// TIA Portal V17 export
// export: Created 2022-06-16T09:21:07.0995622Z, ExportSetting WithDefaults, DisplayName Totally Integrated Automation Portal, DisplayVersion V17, DisplayName TIA Portal Openness, DisplayVersion V17, DisplayName TIA Portal Version Control Interface, DisplayVersion V17, DisplayName STEP 7 Professional, DisplayVersion V17, DisplayName STEP 7 Safety, DisplayVersion V17, DisplayName WinCC Advanced, DisplayVersion V17
DATA_BLOCK "projectParam"   // DB1
{ S7_Optimized_Access := 'TRUE' }
VERSION : 0.1
// stored: AutoNumber true, DBAccessibleFromOPCUA true, IsOnlyStoredInLoadMemory false, IsRetainMemResEnabled false, IsWriteProtectedInAS false, MemoryReserve 100
   VAR
      armParams : Array[1..3] of "typeArmParam";
   END_VAR
BEGIN
   armParams[1..3].armType := 'RCMA';
   armParams[1..3].armGeom.outLength := 8.839;
   armParams[1..3].armGeom.inLength := 9.449;
   armParams[1..3].armGeom.brHeight := 10.47;
   armParams[2].armGeom.brWidth := 10.47;
   armParams[1].motionControlParam.angleInputParam.filterTimeConsts[1..3] := 0.1;
   armParams[2].motionControlParam.angleInputParam.filterTimeConsts[1..3] := 0.1;
   armParams[3].motionControlParam.angleInputParam.filterTimeConsts[1..3] := 0.1;
   armParams[1].motionControlParam.angleInputParam.scalingParams[1].axisNum := 1;
   armParams[1].motionControlParam.angleInputParam.scalingParams[2].axisNum := 2;
   armParams[1].motionControlParam.angleInputParam.scalingParams[3].axisNum := 3;
   armParams[2].motionControlParam.angleInputParam.scalingParams[1].axisNum := 1;
   armParams[2].motionControlParam.angleInputParam.scalingParams[2].axisNum := 2;
   armParams[2].motionControlParam.angleInputParam.scalingParams[3].axisNum := 3;
   armParams[3].motionControlParam.angleInputParam.scalingParams[1].axisNum := 1;
   armParams[3].motionControlParam.angleInputParam.scalingParams[2].axisNum := 2;
   armParams[3].motionControlParam.angleInputParam.scalingParams[3].axisNum := 3;
   armParams[1].motionControlParam.angleInputParam.scalingParams[1..3]."a" := 1.0;
   armParams[2].motionControlParam.angleInputParam.scalingParams[1..3]."a" := 1.0;
   armParams[3].motionControlParam.angleInputParam.scalingParams[1..3]."a" := 1.0;
   armParams[1].motionControlParam.remoteInputParam.easyScalingParams[1].axisNum := 1;
   armParams[1].motionControlParam.remoteInputParam.easyScalingParams[2].axisNum := 2;
   armParams[1].motionControlParam.remoteInputParam.easyScalingParams[3].axisNum := 3;
   armParams[2].motionControlParam.remoteInputParam.easyScalingParams[1].axisNum := 1;
   armParams[2].motionControlParam.remoteInputParam.easyScalingParams[2].axisNum := 2;
   armParams[2].motionControlParam.remoteInputParam.easyScalingParams[3].axisNum := 3;
   armParams[3].motionControlParam.remoteInputParam.easyScalingParams[1].axisNum := 1;
   armParams[3].motionControlParam.remoteInputParam.easyScalingParams[2].axisNum := 2;
   armParams[3].motionControlParam.remoteInputParam.easyScalingParams[3].axisNum := 3;
   armParams[1].motionControlParam.remoteInputParam.easyScalingParams[1..3]."a" := 1.0;
   armParams[2].motionControlParam.remoteInputParam.easyScalingParams[1..3]."a" := 1.0;
   armParams[3].motionControlParam.remoteInputParam.easyScalingParams[1..3]."a" := 1.0;
   armParams[1].motionControlParam.remoteInputParam.convScalingParams[1].axisNum := 1;
   armParams[1].motionControlParam.remoteInputParam.convScalingParams[2].axisNum := 2;
   armParams[1].motionControlParam.remoteInputParam.convScalingParams[3].axisNum := 3;
   armParams[2].motionControlParam.remoteInputParam.convScalingParams[1].axisNum := 1;
   armParams[2].motionControlParam.remoteInputParam.convScalingParams[2].axisNum := 2;
   armParams[2].motionControlParam.remoteInputParam.convScalingParams[3].axisNum := 3;
   armParams[3].motionControlParam.remoteInputParam.convScalingParams[1].axisNum := 1;
   armParams[3].motionControlParam.remoteInputParam.convScalingParams[2].axisNum := 2;
   armParams[3].motionControlParam.remoteInputParam.convScalingParams[3].axisNum := 3;
   armParams[1].motionControlParam.remoteInputParam.convScalingParams[1..3]."a" := 1.0;
   armParams[2].motionControlParam.remoteInputParam.convScalingParams[1..3]."a" := 1.0;
   armParams[3].motionControlParam.remoteInputParam.convScalingParams[1..3]."a" := 1.0;
   armParams[1].motionControlParam.remoteInputParam.filterTimeConsts[1..3] := 0.1;
   armParams[2].motionControlParam.remoteInputParam.filterTimeConsts[1..3] := 0.1;
   armParams[3].motionControlParam.remoteInputParam.filterTimeConsts[1..3] := 0.1;
   armParams[1].motionControlParam.angularSpeedGains[1..3] := 0.018;
   armParams[2].motionControlParam.angularSpeedGains[1..3] := 0.018;
   armParams[3].motionControlParam.angularSpeedGains[1..3] := 0.018;
   armParams[1].motionControlParam.cartSpeedGains[1..3] := 0.15;
   armParams[2].motionControlParam.cartSpeedGains[1..3] := 0.15;
   armParams[3].motionControlParam.cartSpeedGains[1..3] := 0.15;
   armParams[1].motionControlParam.regulParams[1..3].fOn := 1.0;
   armParams[2].motionControlParam.regulParams[1..3].fOn := 1.0;
   armParams[3].motionControlParam.regulParams[1..3].fOn := 1.0;
   armParams[1].motionControlParam.regulParams[1..3].pOn := 1.0;
   armParams[2].motionControlParam.regulParams[1..3].pOn := 1.0;
   armParams[3].motionControlParam.regulParams[1..3].pOn := 1.0;
   armParams[1].motionControlParam.regulParams[1..3].kP := 0.001;
   armParams[2].motionControlParam.regulParams[1..3].kP := 0.001;
   armParams[3].motionControlParam.regulParams[1..3].kP := 0.001;
   armParams[1].motionControlParam.regulParams[1..3].tI := 0.1;
   armParams[2].motionControlParam.regulParams[1..3].tI := 0.1;
   armParams[3].motionControlParam.regulParams[1..3].tI := 0.1;
   armParams[1].motionControlParam.regulParams[1..3].tD := 0.1;
   armParams[2].motionControlParam.regulParams[1..3].tD := 0.1;
   armParams[3].motionControlParam.regulParams[1..3].tD := 0.1;
   armParams[1].motionControlParam.outputParam.filterTimeConsts[1..3] := 0.1;
   armParams[2].motionControlParam.outputParam.filterTimeConsts[1..3] := 0.1;
   armParams[3].motionControlParam.outputParam.filterTimeConsts[1..3] := 0.1;
   armParams[1..3].motionControlParam.satParam.deltaSatGainNeg := 0.01;
   armParams[1].motionControlParam.satParam.satLevels[1..2] := 1.0;
   armParams[1].motionControlParam.satParam.satLevels[3] := 0.5;
   armParams[2].motionControlParam.satParam.satLevels[1..2] := 1.0;
   armParams[2].motionControlParam.satParam.satLevels[3] := 0.5;
   armParams[3].motionControlParam.satParam.satLevels[1..2] := 1.0;
   armParams[3].motionControlParam.satParam.satLevels[3] := 0.5;
   armParams[1..3].motionControlParam.minSetpoint := 0.05;
   armParams[1..3].motionControlParam.minSpeed := 0.01;
   armParams[1].axisParams[1].axisType := 'direct';
   armParams[1].axisParams[2].axisType := 'double';
   armParams[1].axisParams[3].axisType := 'sheave';
   armParams[2].axisParams[1].axisType := 'direct';
   armParams[2].axisParams[2].axisType := 'double';
   armParams[2].axisParams[3].axisType := 'sheave';
   armParams[3].axisParams[1].axisType := 'direct';
   armParams[3].axisParams[2].axisType := 'double';
   armParams[3].axisParams[3].axisType := 'sheave';
   armParams[1].axisParams[1].cylinderType := 'diff';
   armParams[1].axisParams[2..3].cylinderType := 'sym';
   armParams[2].axisParams[1].cylinderType := 'diff';
   armParams[2].axisParams[2..3].cylinderType := 'sym';
   armParams[3].axisParams[1].cylinderType := 'diff';
   armParams[3].axisParams[2..3].cylinderType := 'sym';
   armParams[1].axisParams[1..3].cylinderDir := 1.0;
   armParams[2].axisParams[1..3].cylinderDir := 1.0;
   armParams[3].axisParams[1..3].cylinderDir := 1.0;
   armParams[1].axisParams[1].pistonDiam := 0.1;
   armParams[1].axisParams[2].pistonDiam := 0.14;
   armParams[1].axisParams[3].pistonDiam := 0.11;
   armParams[2].axisParams[1].pistonDiam := 0.1;
   armParams[2].axisParams[2].pistonDiam := 0.14;
   armParams[2].axisParams[3].pistonDiam := 0.11;
   armParams[3].axisParams[1].pistonDiam := 0.1;
   armParams[3].axisParams[2].pistonDiam := 0.14;
   armParams[3].axisParams[3].pistonDiam := 0.11;
   armParams[1].axisParams[1].rodDiam := 0.045;
   armParams[1].axisParams[2].rodDiam := 0.065;
   armParams[1].axisParams[3].rodDiam := 0.055;
   armParams[2].axisParams[1].rodDiam := 0.045;
   armParams[2].axisParams[2].rodDiam := 0.065;
   armParams[2].axisParams[3].rodDiam := 0.055;
   armParams[3].axisParams[1].rodDiam := 0.045;
   armParams[3].axisParams[2].rodDiam := 0.065;
   armParams[3].axisParams[3].rodDiam := 0.055;
   armParams[1].axisParams[1].stroke := 0.62;
   armParams[1].axisParams[2].stroke := 1.4;
   armParams[1].axisParams[3].stroke := 1.0;
   armParams[2].axisParams[1].stroke := 0.62;
   armParams[2].axisParams[2].stroke := 1.4;
   armParams[2].axisParams[3].stroke := 1.0;
   armParams[3].axisParams[1].stroke := 0.62;
   armParams[3].axisParams[2].stroke := 1.4;
   armParams[3].axisParams[3].stroke := 1.0;
   armParams[1].axisParams[1].rodPivotPos[1] := 0.435;
   armParams[1].axisParams[1].rodPivotPos[2] := 0.05;
   armParams[2].axisParams[1].rodPivotPos[1] := 0.435;
   armParams[2].axisParams[1].rodPivotPos[2] := 0.05;
   armParams[3].axisParams[1].rodPivotPos[1] := 0.435;
   armParams[3].axisParams[1].rodPivotPos[2] := 0.05;
   armParams[1].axisParams[1].bodyPivotPos[1] := 0.224;
   armParams[1].axisParams[1].bodyPivotPos[2] := 0.775;
   armParams[2].axisParams[1].bodyPivotPos[1] := 0.224;
   armParams[2].axisParams[1].bodyPivotPos[2] := 0.775;
   armParams[3].axisParams[1].bodyPivotPos[1] := 0.224;
   armParams[3].axisParams[1].bodyPivotPos[2] := 0.775;
   armParams[1].axisParams[1].movingCylinder := TRUE;
   armParams[2].axisParams[1].movingCylinder := TRUE;
   armParams[3].axisParams[1].movingCylinder := TRUE;
   armParams[1].axisParams[1..3].presDrop := 1000000.0;
   armParams[2].axisParams[1..3].presDrop := 1000000.0;
   armParams[3].axisParams[1..3].presDrop := 1000000.0;
   armParams[1].axisParams[1].nomFlow := 1.67E-05;
   armParams[1].axisParams[2].nomFlow := 0.00013;
   armParams[1].axisParams[3].nomFlow := 7.5E-05;
   armParams[2].axisParams[1].nomFlow := 1.67E-05;
   armParams[2].axisParams[2].nomFlow := 0.00013;
   armParams[2].axisParams[3].nomFlow := 7.5E-05;
   armParams[3].axisParams[1].nomFlow := 1.67E-05;
   armParams[3].axisParams[2].nomFlow := 0.00013;
   armParams[3].axisParams[3].nomFlow := 7.5E-05;
   armParams[1].axisParams[1..3].setpointJump := 0.2;
   armParams[2].axisParams[1..3].setpointJump := 0.2;
   armParams[3].axisParams[1..3].setpointJump := 0.2;
   armParams[1].axisParams[1..3].setpointMin := 0.01;
   armParams[2].axisParams[1..3].setpointMin := 0.01;
   armParams[3].axisParams[1..3].setpointMin := 0.01;
   armParams[1].axisParams[2].sheaveDiam := 1.0;
   armParams[1].axisParams[3].sheaveDiam := 0.82;
   armParams[2].axisParams[2].sheaveDiam := 1.0;
   armParams[2].axisParams[3].sheaveDiam := 0.82;
   armParams[3].axisParams[2].sheaveDiam := 1.0;
   armParams[3].axisParams[3].sheaveDiam := 0.82;
   armParams[1].axisParams[1..3].naturalFrequency := 2.0;
   armParams[2].axisParams[1..3].naturalFrequency := 2.0;
   armParams[3].axisParams[1..3].naturalFrequency := 2.0;
   armParams[1].axisParams[1..3].damping := 0.2;
   armParams[2].axisParams[1..3].damping := 0.2;
   armParams[3].axisParams[1..3].damping := 0.2;
END_DATA_BLOCK
